TYPE ST_TTC_6_0 :
(**************************************************************************************
 * 	Application		:	BoxControl Framework
 *	Revision		:	$Revision: 404529 $
 *	Revision date	:	$Date: 2018-04-23 08:21:38 +0200 (Mo., 23 Apr 2018) $
 *	Last changed by	:	$Author: b7bolm $
 *	URL				:	$URL: http://almscdc.swisslog.com/repo/SWPD/Development/BoxControlFramework/20_Release/trunk/01_Software/BCF/BCF/JumpStart/20_Product/10_App/11_Com/10_Lib/10_Conv/12_MFCS/11_SIS/01_DUTs/10_SIS_6_0/ST_TTC_6_0.TcDUT $
 *
 *	Purpose			:	TTC Structure
 *
 * ------------------------------------------------------------------------------------
 *	Copyright Swisslog [IP AG], Switzerland. All rights reserved.
 * 
 * ------------------------------------------------------------------------------------
 *	
 * 	Revision History: 
 *
 * 	VERSION			DATE			INITIALS			DESCRIPTION
 *	0.1				01.01.2001		swl					Example
 *
 **************************************************************************************)
STRUCT
	Position				: STRING(SIS_6_0.POSITION_STRINGLENGTH); // 12 Digit SIS Location MM-GGG-EEEE-FF-Z 
	TU_DataIndex			: STRING(SIS_6_0.TU_DATAINDEX_STRINGLENGTH); // 6 Digit Tu Index
	MsgSequence				: STRING(SIS_6_0.MSG_SEQUENCE_STRINGLENGTH); // 3 Digit Msg Sequence
	TU_ID					: STRING(SIS_6_0.TU_ID_STRINGLENGTH); // 18 Digit SSID 
	AssignmentID			: STRING(SIS_6_0.ASSIGNMENT_ID_STRINGLENGTH); // 8 Digit assignment
	ReturnCode				: STRING(SIS_6_0.ERRORCODE_STRINGLENGTH); // 4 Digit error code
END_STRUCT
END_TYPE

(* stored: Version 1.1.0.1, ProductVersion 3.1.4022.12
   DUT ST_TTC_6_0: Id {ead8227d-275c-4730-b4b4-37828fc7c953} *)
